# EPICS substitutions: MyProject/MyProjectApp/Db/user.substitutions
# SPDX-FileCopyrightText: 2006 Argonne National Laboratory
#
# SPDX-License-Identifier: EPICS

file "db/vacuum.db" {
    { user = "bradm" }
}

file "db/rf.db" {
    { user = "bradm" }
}

file "db/cryo.db" {
    { user = "bradm" }
}

file "db/beam_dump.db" {
    { user = "bradm" }
}

file "db/tungsten_target.db" {
    { user = "bradm" }
}
